// TIA Portal V16 export
// export: Created 2023-03-29T11:03:30.3674306Z, ExportSetting WithDefaults, DisplayName Totally Integrated Automation Portal, DisplayVersion V16 Update 6, DisplayName TIA Portal Version Control Interface, DisplayVersion V16 Update 2, DisplayName TIA Portal Openness, DisplayVersion V16 Update 6, DisplayName STEP 7 Professional, DisplayVersion V16 Update 6, DisplayName STEP 7 Safety, DisplayVersion V16, DisplayName WinCC Advanced, DisplayVersion V16 Update 6
FUNCTION "Kasowanie alarów" : Void   // FC9, LAD
{ S7_Optimized_Access := 'TRUE' }
AUTHOR : rtecmer
VERSION : 0.1
// (*
// //=============================================================================
// //(JZWiK S.A Radosław Tecmer)
// //(c)Copyright (2022) All Rights Reserved
// //-----------------------------------------------------------------------------
// //Testowane z:   (system docelowy z  FW 4.4)
// //Pakiet inżynierski:   TIA Portal (V16 Update 5)
// //Ograniczenia:  ( - )
// //Wymagania:  (minimalne S7-1200 CPU 1215C FW 4.2 .)
// //Funkcjonalnośc: (Kasowanie alarmów napedów przez HMI )
// //-----------------------------------------------------------------------------
// //Zmainy wprowadzone:
// //Wersja  Data       Osoba wprowadzająca zmiany - ekspert
// //01.00.00 09.03.2022 (Tecmer Radosław - twórca) Pieresza wersja 01.00.00
// //=============================================================================
// *)
// stored: AutoNumber true, IsIECCheckEnabled false, SetENOAutomatically false, UDAEnableTagReadback false
BEGIN

REGION Network 2 (SCL): Kasowanie alarmu Z10
   IF  "dbtags_Sterowanie".HMI.resetScreen_1 = TRUE THEN
     // Statement section IF
     IF "Hbit_Alarm_Z10" THEN
       // ustaw reset bit 
        %DB10. := TRUE;
       ;
     END_IF;
     IF "Hbit_Alarm_Z9" THEN
       // ustaw reset bit 
       %DB10. := TRUE;
       ;
     END_IF;

     // kasowanie momentu
     "setAlarm_Moment_Z_9" := FALSE;
     "setAlarm_Moment_Z_10" := FALSE;

     %DB10. := FALSE;
     %DB10. := FALSE;


     ;
   END_IF;

   //IF %DB10.DBX24.0 = FALSE THEN
     // Statement section IF
    // "dbtags_Sterowanie".HMI.resetScreen_1 := False;
   //  %DB10.DBX25.6 := FALSE;

   //  ;
   //END_IF;
END_REGION

REGION Network 3 (SCL): Kasowanie alarmu Z1 Z2
   IF "dbtags_Sterowanie".HMI.resetScreen_5 = TRUE THEN
     // Statement section IF
     IF "Hbit_Alarm_Z1" THEN
       // ustaw reset bit 
       %DB10. := TRUE;
       ;
     END_IF;
     IF "Hbit_Alarm_Z2" THEN
       // ustaw reset bit 
       %DB10. := TRUE;
       ;
     END_IF;


    // kasowanie momentu
     "setAlarm_Moment_Z_1" := FALSE;
     "setAlarm_Moment_Z_2" := FALSE;

     %DB10. := FALSE;
     %DB10. := FALSE;
     ;
   END_IF;
END_REGION

REGION Network 4 (SCL): Kasowanie alarmu Z3 Z4
   IF "dbtags_Sterowanie".HMI.resetScreen_4 = TRUE THEN
     // Statement section IF
     IF "Hbit_Alarm_Z3" THEN
       // ustaw reset bit 
       %DB10. := TRUE;
       ;
     END_IF;
     IF "Hbit_Alarm_Z4" THEN
       // ustaw reset bit 
       %DB10. := TRUE;
       ;
     END_IF;

     // kasowanie momentu
     "setAlarm_Moment_Z_3" := FALSE;
     "setAlarm_Moment_Z_4" := FALSE;

     %DB10. := FALSE;
     %DB10. := FALSE;
     ;
   END_IF;
END_REGION

REGION Network 5 (SCL): Kasowanie alarmu Z5 Z6
   IF "dbtags_Sterowanie".HMI.resetScreen_3 = TRUE THEN
     // Statement section IF
     IF "Hbit_Alarm_Z5" THEN
       // ustaw reset bit 
       %DB10. := TRUE;
       ;
     END_IF;
     IF "Hbit_Alarm_Z6" THEN
       // ustaw reset bit 
       %DB10. := TRUE;
       ;
     END_IF;

     // kasowanie momentu
     "setAlarm_Moment_Z_5" := FALSE;
     "setAlarm_Moment_Z_6" := FALSE;

     %DB10. := FALSE;
     %DB10. := FALSE;

     ;
   END_IF;
END_REGION

REGION Network 6 (SCL): Kasowanie alarmu Z7 Z8
   IF "dbtags_Sterowanie".HMI.resetScreen_2 = TRUE THEN
     // Statement section IF
     IF "Hbit_Alarm_Z7" THEN
       // ustaw reset bit 
       %DB10. := TRUE;
       ;
     END_IF;
     IF "Hbit_Alarm_Z8" THEN
       // ustaw reset bit 
       %DB10. := TRUE;
       ;
     END_IF;

     // kasowanie momentu
     "setAlarm_Moment_Z_7" := FALSE;
     "setAlarm_Moment_Z_8" := FALSE;

     %DB10. := FALSE;
     %DB10. := FALSE;

     ;
   END_IF;
END_REGION

REGION Network 11: Kasowanie alarmu Z1 Z2
END_REGION
END_FUNCTION
